FUNCTION_BLOCK IO_DI (* Digital input primitive; Backend 0 simulated, 1 GPIO (IX + GPIOChip handle), 2 Modbus CLIENT *)
  (* Standard: 61499-2 *)
  (* Version 2.0, 2026-09-27, Project contributors, Filling cell reference model *)
  PACKAGE fillingcell;
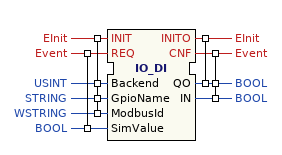
  EVENT_INPUT
    INIT : EInit WITH Backend, GpioName, ModbusId;
    REQ WITH SimValue;
  END_EVENT
  EVENT_OUTPUT
    INITO : EInit WITH QO;
    CNF WITH QO, IN;
  END_EVENT
  VAR_INPUT
    Backend : USINT;
    GpioName : STRING;
    ModbusId : WSTRING;
    SimValue : BOOL;
  END_VAR
  VAR_OUTPUT
    QO : BOOL;
    IN : BOOL;
  END_VAR
  FBS
    Route : fillingcell::IO_RouteDI;
    Gpio : eclipse4diac::io::IX;
    Bus : iec61499::net::CLIENT_0_1;
  END_FBS
  EVENT_CONNECTIONS
    INIT TO Route.INIT;
    Route.INIT_IO TO Gpio.INIT;
    Gpio.INITO TO Bus.INIT;
    Bus.INITO TO Route.IO_READY;
    Route.INITO TO INITO;
    REQ TO Route.REQ;
    Route.REQ_G TO Gpio.REQ;
    Route.REQ_M TO Bus.REQ;
    Gpio.CNF TO Route.CNF_G;
    Bus.CNF TO Route.CNF_M;
    Route.CNF TO CNF;
  END_CONNECTIONS
  DATA_CONNECTIONS
    Backend TO Route.Backend;
    GpioName TO Gpio.PARAMS;
    ModbusId TO Bus.ID;
    Route.GQI TO Gpio.QI;
    Route.MQI TO Bus.QI;
    Gpio.QO TO Route.QO_G;
    Bus.QO TO Route.QO_M;
    Route.QO TO QO;
    SimValue TO Route.SimValue;
    Gpio.IN TO Route.IN_G;
    Bus.RD_1 TO Route.IN_M;
    Route.IN TO IN;
  END_CONNECTIONS
END_FUNCTION_BLOCK
